// TIA Portal V19 export
FUNCTION "PB_ChainWash" : Void   // FC93, STL
TITLE = Pb - Chain wash
{ S7_Optimized_Access := 'TRUE' }
NAME : PBLYECIP
VERSION : 0.0
// Comment
// stored: AutoNumber false
   VAR_TEMP
      alarmbit : Int;
   END_VAR
BEGIN

NETWORK
TITLE = 
// Comment Flash K9 when filler ready for CIP
      A     "CHAIN_WASH";
      AN    "S0 CIP TANK";
      AN    "S0 FILLER";
      AN    "S0 CHAIN WASH";
      R     "LEDAssignment".K10_LIGHT;  // "LIGHT_K10_CHAIN"
      S     "LEDAssignment".K10_FLASH;  // "FLASH_K10_CHAIN"
      JC    B001;

      AN    "CHAIN_WASH";
      R     "LEDAssignment".K10_LIGHT;  // "LIGHT_K10_CHAIN"
      R     "LEDAssignment".K10_FLASH;  // "FLASH_K10_CHAIN"
B001: NOP   0;

NETWORK
TITLE = 
// Comment Blocing
      AN    "CHAIN_WASH";  // CHAIN WASH SIGNAL MISSING
      A     "S0 CHAIN WASH";
      JC    C001;  // STOP CIP

      AN    "LEDAssignment".K10_BUTTON;  // "PbK10CHAINWASH"            // START/STOP CIP FILLER
      BEC;
      R     "LEDAssignment".K10_BUTTON;  // "PbK10CHAINWASH"

      A     "S0 CHAIN WASH";
      JC    C001;  // STOP CIP

      A     "S0 CIP TANK";
      S     "ProcessAndPbAlarms"."A"[14];  //A14_CipOnTankStared// CIP TANK STARTED
      L     14;
      JC    Alrm;
//      BEC

      A     "S0 FILLER";
      S     "ProcessAndPbAlarms"."A"[7];  //A07_CipUnitOccupied//CIP_UNIT_OCCUIPED
      L     7;
      JC    Alrm;
//      BEC

      AN    "PA0572_Air";
      S     "ProcessAndPbAlarms"."A"[3];  //A03_NoInstrumentAir// no intrument air
      L     3;
      JC    Alrm;
//      BEC

      AN    "PA0561_Steam";
      S     "ProcessAndPbAlarms"."A"[4];  //A04_NoSteam// no steam
      L     4;
      JC    Alrm;
//      BEC
      S     "S0 CHAIN WASH";
      S     "LEDAssignment".K10_FLASH;  // "FLASH_K10_CHAIN"
      S     "LEDAssignment".K10_LIGHT;  // "LIGHT_K10_CHAIN"
      BEU;

C001: R     "S0 CHAIN WASH";
      R     "LEDAssignment".K10_FLASH;  //  "FLASH_K10_CHAIN"
      R     "LEDAssignment".K10_LIGHT;  // "LIGHT_K10_CHAIN"
      R     "AutoTT0172/IP0157";
      R     "MY0158";
      R     "MM0139";
      R     "MY0114";  // drain
      R     "MY0115";
      R     "MY0116";
      R     "MY0117";
      R     "MY0119";
      R     "CONTROL CIP TANK";
      BEU;

NETWORK
TITLE = Blockings alarm text
// Blockings alarm
Alrm: NOP   1;
      T     #alarmbit;
      CALL  "Set_Pop_Up_Blocking"
      ( alarmTextNum := #alarmbit
      );  // start blockings text


END_FUNCTION
